TYPE HydraulicsTabs :
(
	OVERVIEW := 0,
    TECHNICAL := 1,
    IO := 2,
    CONFIG := 3
);
END_TYPE

(* stored: Version 1.1.0.1, ProductVersion 3.1.4018.5
   DUT HydraulicsTabs: Id {39543a4c-70ec-4316-87b9-a8ce565217b4} *)
